// TIA Portal V20 export
// export: Created 2025-12-01T14:56:17.7317213Z, ExportSetting None, DisplayName Totally Integrated Automation Portal, DisplayVersion V20 Update 3, DisplayName TIA Portal Openness, DisplayVersion V20 Update 3, DisplayName TIA Portal Version Control Interface, DisplayVersion V20 Update 3, DisplayName STEP 7 Professional, DisplayVersion V20 Update 3, DisplayName STEP 7 Safety, DisplayVersion V20 Update 2, DisplayName WinCC Basic/Comfort/Advanced, DisplayVersion V20 Update 3, DisplayName WinCC Professional, DisplayVersion V20 Update 3, DisplayName WinCC Unified, DisplayVersion V20 Update 3
TYPE "UDT_HMI_LineaPotencia"
   STRUCT
      Proteccion : Bool;   // Estado de la Proteción Magnetico Termica Diferencial
      Bit_01 : Bool;   // Reserva
      FeedBackContactor : Bool;   // Retro-Alimentación de reles y contactores para activación de la linea
      ActivacionContactor : Bool;   // Estado de la Salida del PLC para activación del rele
      Bit_04 : Bool;   // Reserva
      PilotoRojo : Bool;   // Piloto Rojo --> Linea sin Tension
      PilotoVerde : Bool;   // Piloto Verde --> Linea en Tension
      ErrorFeedBack : Bool;   // Error de FeedBack
      Bit_10 : Bool;   // Reserva
      Bit_11 : Bool;   // Reserva
      EsperaActivacion : Bool;   // Linea en Espera de Turno de Activación
      CondicionesActivacion : Bool;   // Condiciones necesarias para activación de Linea
      Bit_14 : Bool;   // Reserva
      Bit_15 : Bool;   // Reserva
      Bit_16 : Bool;   // Reserva
      Bit_17 : Bool;   // Reserva
   END_STRUCT;
END_TYPE
